Universal Robots PolyScope program: andrea14.urp

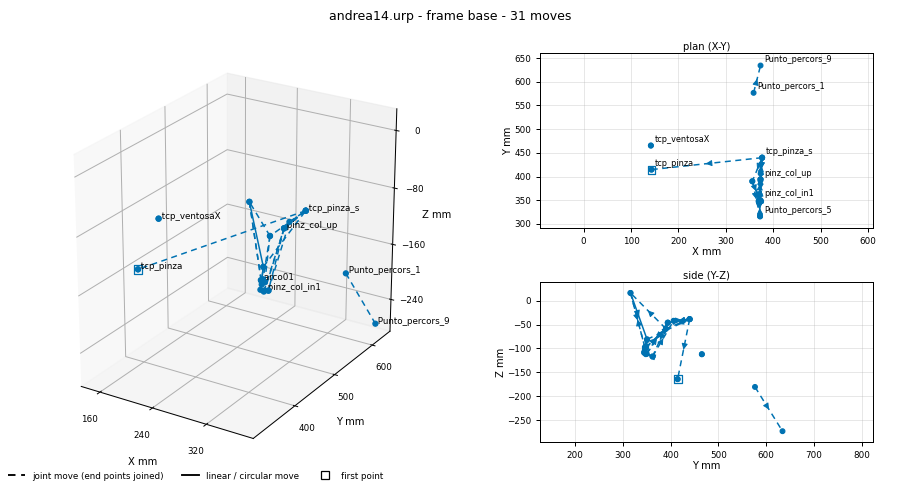
[picture p0: tool path of andrea14.urp in frame base, 31 of 53 moves have a stored position in this frame; points joined in program order, loops and branches not executed]
Program andrea14 (installation=Kong_install12 directory=/programs/usbdisk/andrea14 createdIn=3.15.4.106291 lastSavedIn=3.15.4.106291 robotSerialNumber=2017357596)
Calibrated DH parameters: a=[0.000104, -0.381245, -0.385946, 0.00002, 0.000083, 0]; d=[0.089177, 59.99214, -36.297918, -23.584132, 0.094784, 0.082552]; alpha=[1.570197, -0.003145, 0.002952, 1.570494, -1.570091, 0]; deltaTheta=[-0.00001, -0.459739, 0.638868, -0.17972, -0.000006, -0.000462]
InitVariablesNode variables(variable(name=XY, expression=[0,0]), variable(name=ant, expression=3), variable(name=col, expression=4), variable(name=dump, expression=5), variable(name=ghr, expression=2), variable(name=nCycle, expression=0), variable(name=nfc, expression=1), variable(name=pallStocks, expression=[16,16,16,40,16,16,16,40,16,16,16,40,16,40,0,0,0,0,0,0,0,0,0,0]), variable(name=pick, expression=[0,0]))
Robot Program (runOnlyOnce=false)
  Script file /programs/Kong/relPose.script
    | def relPose(FeaturePose,vect):
    | 
    |     # FeaturePose is the pose for the feature
    |     # vect = p[0.1, 0, 0, 0, 0, 0] makes us move 10cm in the X direction of the feature
    |     # credits: https://forum.universal-robots.com/t/move-tcp-relative-to-feature/15492
    | 
    |    PoseRelativeToFeature = pose_trans(pose_inv(FeaturePose), get_actual_tcp_pose())
    |    MoveTCPRelativeToFeature = pose_add(PoseRelativeToFeature, vect)
    |    return pose_trans(FeaturePose, MoveTCPRelativeToFeature)
    | 
    | end
  Script file /programs/Kong/totf.script_bak
    | def totf(tcpf):
    | 
    |     return sqrt(tcpf[0]*tcpf[0]+tcpf[1]*tcpf[1]+tcpf[2]*tcpf[2]+tcpf[3]*tcpf[3]+tcpf[4]*tcpf[4]+tcpf[5]*tcpf[5])
    | 
    | end
  Script file /programs/Kong/tcpMov.script
    | def tcpMov(vect):
    | 
    |     # FeaturePose is the pose for the feature
    |     # vect = p[0.1, 0, 0, 0, 0, 0] makes us move 10cm in the X direction of the feature
    |     # credits: https://forum.universal-robots.com/t/move-tcp-relative-to-feature/15492
    | 
    |    tcp_pose = get_actual_tcp_pose()
    |    return pose_add(tcp_pose, vect)
    | 
    | 
    | end
  Script file /programs/Kong/calcItemPosition.script_bak
    | def calcItemPosition(pick, item, pallDefs, grid, featOrigin):
    | 
    |     # calcola la posizione assoluta del pezzo scelto da pickPalletItem
    | 
    |     # nPosX è il numero di colonne
    |     # nPosY è il numero di righe
    |     # distX è la distanza tra colonne
    |     # distY è la distanza tra righe
    |     # [posX1, posY1] è la posizione del primo pezzo rispetto all'origine del pallet
    | 
    |     nPallet = pick[0] + 1 # numero del pallet (gli id partono da 0)
    |     nItem = pick[1] + 1 # numero del pezzo
    | 
    |     nPosXgrid = grid[0] # numero di posizioni della giglia in X
    |     distXgrid = grid[2] # distanza tra gli slot della griglia in X
    |     distYgrid = grid[3] # distanza tra gli slot della griglia in Y
    | 
    |     pallPosX = nPallet%nPosXgrid
    |     if(pallPosX==0): pallPosX = nPosXgrid end
    |     pallPosY = ceil(nPallet/nPosXgrid)
    | 
    |     pallPosX1 = grid[4]
    |     pallPosY1 = grid[5]
    | 
    | 
    |     nPosX = pallDefs[item,0]
    |     nPosY = pallDefs[item,1]
    |     distX = pallDefs[item,2]
    |     distY = pallDefs[item,3]
    |     posX1 = pallDefs[item,4]
    |     posY1 = pallDefs[item,5]
    | 
    |     posX = nItem%nPosX
    |     if(posX==0): posX = nPosX end
    |     posY = ceil(nItem/nPosX)
    | 
    |     # [X,Y] è la posizione del pezzo rispetto all'origine della griglia
    | 
    |     X=distX*(posX - 1) + posX1 + distXgrid*(pallPosX - 1) + pallPosX1
    |     Y=distY*(posY - 1) + posY1 + distYgrid*(pallPosY - 1) + pallPosY1
    |     xy=[X,Y]
    | 
    |     return xy
    | 
    |  end
  Script file /programs/usbdisk/andrea8/pickPalletItem.script
    | def pickPalletItem(type, pallDefs, pallTypes, pallStocks):
    | 
    |   # seleziona un pezzo sulla griglia, noti il tipo di pezzo e lo stato della griglia
    | 
    |   # lo script funziona finché le variabili del robot non vengono resettate. Tuttavia, anche
    |   # in caso di riavvio, è possibile scrivere manualmente le info sulla griglia e lo stock
    |   # all'inizio del programma, così da 'insegnare' al robot dove farlo
    |   # riprendere
    | 
    |   iPallet = 0 # inizializzo l'id del pallet
    | 
    |   while iPallet < length(pallStocks):
    | 
    |     if pallTypes[iPallet] == type and pallStocks[iPallet] > 0 :
    | 
    |       nItems = pallStocks[iPallet] # numero di pezzi nello stock del pallet iesimo
    | 
    |       nPosX = pallDefs[type,0] # numero di posizioni lungo x, come definito per il pallet di tipo "type"
    |       nPosY = pallDefs[type,1] # numero di posizioni lungo y, come definito per il pallet di tipo "type"
    | 
    |       stockMax = nPosX*nPosY
    |       iItem = stockMax - nItems # id del pezzo
    | 
    |       pick = [iPallet,iItem]
    | 
    |       # pick = [id del pallet, id del pezzo]
    | 
    |       return pick
    |  end
    | iPallet = iPallet + 1
    | end
    | end
  Script file /home/ur/ursim-current/programs/andrea11/stockUpdate.script_bak
    | def stockUpdate(pick,stock):
    | 
    |     # simple function that ingests the output of pickItem and returns the
    |     # modified stock array. just so to avoid using global variables and
    |     # multi-dimensional arrays
    | 
    |     i = pick[0]
    |     stock[i] = stock[i] - 1
    |     return stock
    | 
    | 
    | end
  Script file /programs/Kong/ini_grid.script_bak.script
    | def ini_grid():
    | 
    |     # grid = [nPallPosX, nPallPosY, distPallX, distPallY, pallPosX1, pallPosY1, pallPosZ1]
    |     # la struttura e' del tutto analoga in logica con quella espressa in defs
    |     grid = [4, 4, 90, 90, 10, 20, 6]
    |     return grid
    | end
  Script file /programs/Kong/ini_defs.script
    | def ini_defs():
    | 
    |     # definition = [nPosX,nPosY,distX,distY,posX1,posY1,posZ1]
    | 
    |     # nPosX è il numero di colonne
    |     # nPosY è il numero di righe
    |     # distX è la distanza tra colonne
    |     # distY è la distanza tra righe
    |     # [posX1, posY1] è la posizione del primo pezzo rispetto all'origine del pallet
    |     # posZ1 e' la posizione che deve raggiungere il TCP lungo asse Z, che sarebbe asse verticale
    | 
    |     defs = [
    |         [0, 0, 0, 0, 0, 0, 0], # slot vuoto
    |         [4, 10, 18, 8, 12, 7.4, 9.1], # pallet nfc
    |         [4, 4, 21, 21, 8.2, 7.5, 50], # pallet ghiere
    |         [1, 1, 0, 0, 132.06, 44, 16.05], # stazione antenna
    |         [1, 2, 0, 40, 20.256, 24, 27.85], # stazione incollaggio
    |         [1, 1, 0, 0, 40, 40, 50] # cestino
    |     ]
    |     return defs
    | end
  Script file /programs/Kong/ini_types.script_bak_bak
    | def ini_types():
    | 
    |     visualTypes = [
    | 
    |         [0, 0, 0, 0],
    |         [0, 0, 0, 0],
    |         [0,0,0,0],
    |         [0,0,0,0],
    |         [0,ghr,0,nfc],
    |         [dump,0,0,0]
    | 
    |     ]
    | 
    | # purtroppo fare questa array vuota di dimensione (righe)x(colonne) per aggirare le limitazioni di UR
    | # bisogna ricordarsi di cambiare questa dichiarazione di types se si cambia dimensione griglia
    | 
    |      types = [0,0,0,0,0,0,0,0,0,0,0,0,0,0,0,0,0,0,0,0,0,0,0,0]
    | 
    |     iii = 0
    |     s = size(visualTypes)
    |     i = 0
    |     while i < s[0]:
    | 
    |         ii=0
    |         while ii < s[1]:
    | 
    |             types[iii] = visualTypes[s[0]-1-i,ii]
    |             ii = ii + 1
    |             iii = iii + 1
    |         end
    |     i = i + 1
    |     end
    |     return types
    | end
  Script file /programs/Kong/ini_stocks2.script
    | def ini_stocks(defs, types):
    | 
    |     global f = -1 # usa questo carattere per inizializzare automaticamente pallet pieni
    | 
    |     visualStocks = [
    | 
    |         [f, f, f, f],
    |         [f, f, f, f],
    |         [f, f, f, f],
    |         [f, f, f, f],
    |         [f, f, f, 27],
    |         [f ,f, f, f]
    | 
    |     ]
    | 
    | # purtroppo fare questa array vuota di dimensione (righe)x(colonne) per aggirare le limitazioni di UR
    | # bisogna ricordarsi di cambiare questa dichiarazione di types se si cambia dimensione griglia
    | 
    |      stocks = [0,0,0,0,0,0,0,0,0,0,0,0,0,0,0,0,0,0,0,0,0,0,0,0]
    | 
    |     iii = 0
    |     s = size(visualStocks)
    |     i = 0
    |     while i < s[0]:
    | 
    |         ii=0
    |         while ii < s[1]:
    |             if visualStocks[s[0]-1-i,ii] == f:
    |                 nPosX = defs[types[iii], 0]
    |                 nPosY = defs[types[iii], 1]
    |                 stocks[iii] = nPosX*nPosY
    |             else:
    | 
    |                 stocks[iii] = visualStocks[s[0]-1-i,ii]
    |             end
    |             ii = ii + 1
    |             iii = iii + 1
    |         end
    |     i = i + 1
    |     end
    |     return stocks
    | end
  Script file /programs/Kong/gen_tcp_grid.script
    | def next_tcp_grid_pos(cur_pos,size,dist):
    | 
    | # size e' la dimensione della griglia da generare,
    | # 2 significa 2x2, 3 significa 3x3 etc
    | 
    | rel_p = [0,0]
    | tcpp = get_actual_tcp_pose()
    | 
    | posX = cur_pos%size
    | if(posX==0): posX = size end
    | posY = ceil(cur_pos/size)
    | 
    | actual_dx = -dist*(size-1)/2 + (posX-1)*dist
    | actual_dy= -dist*(size-1)/2 + (posY-1)*dist
    | 
    | posX = (cur_pos+1)%size
    | if(posX==0): posX = size end
    | posY = ceil((cur_pos+1)/size)
    | 
    | next_dx = -dist*(size-1)/2 + (posX-1)*dist
    | next_dy= -dist*(size-1)/2 + (posY-1)*dist
    | 
    | rel_p = [next_dx - actual_dx, next_dy - actual_dy]
    | 
    | return rel_p
    | 
    | end
  If nCycle≟0
    Set DigitalOutput pin=digital_out[1]; digitalValue=0
    Set DigitalOutput pin=digital_out[0]; digitalValue=0
    pallTypes := ini_types()
    nfc_ck_override := True
    grid := ini_grid()
    pallDefs := ini_defs()
    pallStocks := ini_stocks(pallDefs,pallTypes)
    SuppressedNode
      Popup Message (haltProgram=false inputType=Variable) variable=grid
    ghr := ghr
    nfc := nfc
    ant := ant
    col := col
    dump := dump
    URCap Close Gripper (SCHUNK End-of-Arm Modular System for UR, SCHUNK GmbH & Co.)
    nCycle := 1
    nfc_check := False
    ghr_check := False
    cmp_x_in := 0
    cmp_y_in := 0
    cmp_x_out := 0
    cmp_y_out := 0
    cmp_x := False
    cmp_y := False
    Wait Sleep waitTime=1
  MoveJ speed 60 deg/s, acceleration 80 deg/s^2 (useActiveTCP=false) tcp=Pinza
    Waypoint tcp_pinza: TCP in base x=143.254 y=414.593 z=-164.379 mm, rx=-2.3787 ry=0.7213 rz=1.7106 rad; joints [-127.002, -49.901, 105.969, -114.073, -24.505, -23.784] deg; flange x=184.208 y=554.939 z=9.914 mm, rx=-2.3787 ry=0.7213 rz=1.7106 rad
    item := ghr
    pick := pickPalletItem(item,pallDefs,pallTypes,pallStocks)
    lastpick := pick
    SuppressedNode
      Popup Message (haltProgram=false inputType=Variable) variable=pick
    XY := calcItemPosition(pick, item,pallDefs, grid,piano_moduli)
    p_pall := relPose(piano_moduli,p[(XY[0]+cmp_x_in)/1000,(XY[1]+cmp_y_in)/1000,0.0,0.0,0.0,0.0])
    SuppressedNode
      Popup Message (haltProgram=false inputType=Variable) variable=XY
    Waypoint Punto_percors (Variable): motionParameters(blendRadius=0.004); variable=p_pall
  MoveL speed 250 mm/s, acceleration 1200 mm/s^2 (useActiveTCP=false) tcp=Pinza; feature=Base
    MoveDirectionNode (selectedDirection=ZMinus toolParams=0.05, 1.2) feature=origine_moduli
      Until DISTANCE (allowActions=true deceleration=3 distanceNodeType=STOP) Distance=0.1; motionParameters(blendRadius=0)
        URCap Open Gripper (SCHUNK End-of-Arm Modular System for UR, SCHUNK GmbH & Co.)
        p_pezzo := relPose(piano_moduli,p[0.0, 0.0, 125/1000, 0.0, 0.0, 0.0])
        Waypoint Punto_percors (Variable): variable=p_pezzo
        pallStocks := stockUpdate(pick,pallStocks)
        cmp_x := False
        cmp_y := False
      Until EXPRESSION (allowActions=true) ExpressionBranch=totf(get_tcp_force())>92
        ghr_check := False
        ghr_attpt := 0
        cmp_x := True
        Loop While (checkContinuously=false) expression=ghr_check≟ False
          SuppressedNode
            MoveL speed 125 mm/s, acceleration 600 mm/s^2 (useActiveTCP=false) tcp=Pinza; feature=Base
              p_pezzo := relPose(piano_moduli,p[0.0, 0.0, -125*0.001, 0.0, 0.0, 0.0])
              Waypoint Punto_percors (Variable): variable=p_pezzo
              URCap Open Gripper (SCHUNK End-of-Arm Modular System for UR, SCHUNK GmbH & Co.)
              p_pezzo := relPose(piano_moduli,p[0.0, 0.0, 125/1000, 0.0, 0.0, 0.0])
              Waypoint Punto_percors (Variable): variable=p_pezzo
              pallStocks := stockUpdate(pick,pallStocks)
              SuppressedNode
                Popup Message (haltProgram=false inputType=Variable) variable=pallStocks
          ghr_attpt := ghr_attpt+1
          MoveL speed 125 mm/s, acceleration 600 mm/s^2 (useActiveTCP=false) tcp=Pinza; feature=Base
            Waypoint Punto_percor_14 (Relative): relativeFromPosition TCP in base x=29.478 y=440.875 z=-307.868 mm, rx=-2.3716 ry=0.6969 rz=1.6945 rad; joints [-115.757, -28.156, 105.846, -162.962, -20.903, 4.096] deg; TCP in base x=29.576 y=447.944 z=-300.79 mm, rx=-2.3716 ry=0.6967 rz=1.6945 rad; joints [-115.45, -28.728, 105.08, -162.418, -20.875, 4.938] deg; flange x=68.514 y=584.323 z=-122.922 mm, rx=-2.3716 ry=0.6967 rz=1.6945 rad
          If ghr_attpt≟8
            ghr_attpt := 0
            cmp_y := True
            MoveL speed 50 mm/s, acceleration 500 mm/s^2 (useActiveTCP=false) tcp=Pinza; feature=Base
              Waypoint Punto_percor_15 (Relative): relativeFromPosition TCP in base x=141.409 y=424.504 z=-142.092 mm, rx=-2.3788 ry=0.7214 rz=1.7106 rad; joints [-126.265, -51.639, 104.635, -112.37, -24.118, -22.276] deg; TCP in base x=142.404 y=430.165 z=-147.7 mm, rx=-2.3787 ry=0.7215 rz=1.7107 rad; joints [-126.02, -50.501, 103.739, -113.086, -23.994, -21.754] deg; flange x=183.37 y=570.533 z=26.574 mm, rx=-2.3787 ry=0.7215 rz=1.7107 rad
          MoveL speed 50 mm/s, acceleration 500 mm/s^2 (useActiveTCP=false) tcp=Pinza; feature=Base
            Waypoint Punto_percor_10 (Relative): relativeFromPosition TCP in base x=141.556 y=430.223 z=-147.722 mm, rx=-2.3788 ry=0.7212 rz=1.7106 rad; joints [-125.948, -50.518, 103.824, -113.299, -23.962, -21.607] deg; TCP in base x=141.537 y=429.491 z=-147.044 mm, rx=-2.3788 ry=0.7213 rz=1.7106 rad; joints [-125.989, -50.655, 103.927, -113.183, -23.981, -21.693] deg; flange x=182.477 y=569.847 z=27.245 mm, rx=-2.3788 ry=0.7213 rz=1.7106 rad
          MoveDirectionNode (selectedDirection=ZMinus toolParams=0.05, 1.2) feature=origine_moduli
            Until DISTANCE (allowActions=true deceleration=3 distanceNodeType=STOP) Distance=0.017; motionParameters(blendRadius=0)
              URCap Open Gripper (SCHUNK End-of-Arm Modular System for UR, SCHUNK GmbH & Co.)
              p_pezzo := relPose(piano_moduli,p[0.0, 0.0, 125/1000, 0.0, 0.0, 0.0])
              Waypoint Punto_percors (Variable): variable=p_pezzo
              pallStocks := stockUpdate(pick,pallStocks)
              ghr_check := True
            Until EXPRESSION (allowActions=true) ExpressionBranch=totf(get_tcp_force())>80
              MoveL speed 50 mm/s, acceleration 500 mm/s^2 (useActiveTCP=true) feature=Base
                Waypoint Punto_percors_6 (Relative): relativeFromPosition TCP in base x=4.07 y=674.667 z=69.754 mm, rx=1.9149 ry=-1.1485 rz=-1.8457 rad; joints [-112.275, -36.345, 91.167, -133.706, -10.047, 30.658] deg; TCP in base x=4.143 y=678.166 z=73.281 mm, rx=1.9147 ry=-1.1486 rz=-1.8457 rad; joints [-112.167, -36.367, 90.585, -133.706, -10.021, 31.279] deg; flange x=70.38 y=685.456 z=-8.016 mm, rx=1.9147 ry=-1.1486 rz=-1.8457 rad
  SuppressedNode
    If cmp_x≟ True removedSiblings(If(type=Else checkContinuously=false, children(Assignment(valueSource=Expression, variable=cmp_x_in, expression=cmp_x_in+1))))
      cmp_x_in := cmp_x_in-1
  SuppressedNode
    If cmp_y≟ True removedSiblings(If(type=Else checkContinuously=false, children(Assignment(valueSource=Expression, variable=cmp_y_in, expression=cmp_y_in+1))))
      cmp_y_in := cmp_y_in-1
  nfc_check := False
  Loop While (checkContinuously=false) expression=nfc_check≟ False
    MoveJ speed 60 deg/s, acceleration 80 deg/s^2 (useActiveTCP=false) tcp=Ventosa
      Waypoint tcp_ventosaX: TCP in base x=141.964 y=465.304 z=-112.234 mm, rx=-2.2905 ry=-0.5963 rz=-0.2623 rad; joints [-121.653, -49.489, 100.632, -2.161, 68.856, 127.498] deg; flange x=142.46 y=500.184 z=-13.074 mm, rx=-2.2905 ry=-0.5963 rz=-0.2623 rad
      item := dump
      pick := pickPalletItem(item,pallDefs,pallTypes,pallStocks)
      SuppressedNode
        Popup Message (haltProgram=false inputType=Variable) variable=pick
      XY := calcItemPosition(pick, item,pallDefs, grid,piano_moduli)
      p_pall := relPose(piano_moduli,p[XY[0]/1000,XY[1]/1000,0.0,0.0,0.0,0.0])
      SuppressedNode
        Popup Message (haltProgram=false inputType=Variable) variable=XY
      Waypoint Punto_percors (Variable): motionParameters(blendRadius=0.005); variable=p_pall
      Set DigitalOutput pin=digital_out[0]; digitalValue=0
    MoveJ speed 60 deg/s, acceleration 80 deg/s^2 (useActiveTCP=false) tcp=Ventosa
      Waypoint tcp_ventosaX: TCP in base x=141.964 y=465.304 z=-112.234 mm, rx=-2.2905 ry=-0.5963 rz=-0.2623 rad; joints [-121.653, -49.489, 100.632, -2.161, 68.856, 127.498] deg; flange x=142.46 y=500.184 z=-13.074 mm, rx=-2.2905 ry=-0.5963 rz=-0.2623 rad
      SuppressedNode
        Waypoint tcp_ventosaY_s: TCP in base x=355.984 y=389.916 z=-58.857 mm, rx=-1.401 ry=-1.0647 rz=1.3858 rad; joints [-146.472, -36.177, 73.345, -37.097, -55.375, 194.745] deg; pose in feature x=141.985 y=465.345 z=-112.215 mm, rx=-1.4011 ry=-1.0646 rz=1.3857 rad; flange x=401.93 y=456.119 z=8.64 mm, rx=-1.401 ry=-1.0647 rz=1.3858 rad
      item := nfc
      pick := pickPalletItem(item,pallDefs,pallTypes,pallStocks)
      SuppressedNode
        Popup Message (haltProgram=false inputType=Variable) variable=pick
      XY := calcItemPosition(pick, item,pallDefs, grid,piano_moduli)
      p_pall := relPose(piano_moduli,p[XY[0]/1000,XY[1]/1000,0.0,0.0,0.0,0.0])
      SuppressedNode
        Popup Message (haltProgram=false inputType=Variable) variable=XY
      Waypoint Punto_percors (Variable): variable=p_pall
      p_pezzo := relPose(piano_moduli,p[0.0, 0.0, -170*0.001, 0.0, 0.0, 0.0])
      Waypoint Punto_percors (Variable): variable=p_pezzo
      Set DigitalOutput pin=digital_out[0]; digitalValue=1
    Loop Counting (count=3) loopVariable(name=Ciclo_4)
      MoveL speed 1.5 mm/s, acceleration 5 mm/s^2 (useActiveTCP=false) tcp=Ventosa; feature=Base
        p_pezzo := relPose(piano_moduli,p[0.0, 0.0, -12*0.001, 0.0, 0.0, 0.0])
        Waypoint Punto_percors (Variable): variable=p_pezzo
        Wait Sleep waitTime=4
        p_pezzo := relPose(piano_moduli,p[0.0, 0.0, 12/1000, 0.0, 0.0, 0.0])
        Waypoint Punto_percors (Variable): variable=p_pezzo
        SuppressedNode
          Popup Message (haltProgram=false inputType=Variable) variable=pallStocks
    pallStocks := stockUpdate(pick,pallStocks)
    MoveJ speed 60 deg/s, acceleration 80 deg/s^2 (useActiveTCP=true)
      Waypoint Punto_percor_17 (Relative): relativeFromPosition TCP in base x=284.521 y=550.156 z=-280.841 mm, rx=-2.2786 ry=-0.6987 rz=-0.1736 rad; joints [-129.352, -17.294, 64.16, 9.308, 60.336, 116.033] deg; TCP in base x=285.519 y=620.503 z=-209.796 mm, rx=-2.2786 ry=-0.6987 rz=-0.1734 rad; joints [-125.512, -17.144, 49.814, 21.783, 62.478, 119.625] deg; flange x=285.39 y=658.018 z=-111.601 mm, rx=-2.2786 ry=-0.6987 rz=-0.1734 rad
    MoveJ speed 60 deg/s, acceleration 80 deg/s^2 (useActiveTCP=false) tcp=Ventosa
      Waypoint Punto_percors_1: motionParameters(blendRadius=0.005); TCP in base x=358.691 y=576.543 z=-180.701 mm, rx=-2.2887 ry=-0.6045 rz=-0.2628 rad; joints [-132.678, -21.575, 54.335, 20.288, 61.783, 117.598] deg; flange x=358.684 y=611.454 z=-81.55 mm, rx=-2.2887 ry=-0.6045 rz=-0.2628 rad
      Waypoint Punto_percors_9: TCP in base x=373.356 y=634.147 z=-273.366 mm, rx=-2.2782 ry=-0.6995 rz=-0.1742 rad; joints [-130.565, 2.612, 17.324, 36.849, 59.589, 114.737] deg; flange x=373.138 y=671.629 z=-175.158 mm, rx=-2.2782 ry=-0.6995 rz=-0.1742 rad
    MoveL speed 125 mm/s, acceleration 600 mm/s^2 (useActiveTCP=false) tcp=Ventosa; feature=Base
      p_pezzo := relPose(piano_moduli,p[0.0, 0.0, -60*0.001, 0.0, 0.0, 0.0])
      Waypoint Punto_percors (Variable): variable=p_pezzo
      SuppressedNode
        Wait Sleep waitTime=2.5
      If nfc_ck_override≟ True
        nfc_check := True
      Loop Counting (count=5) loopVariable(name=Ciclo_2)
        Wait Sleep waitTime=0.5
        If digital_in[4]≟ True
          nfc_check := True
      p_pezzo := relPose(piano_moduli,p[0.0, 0.0, 40/1000, 0.0, 0.0, 0.0])
      Waypoint Punto_percors (Variable): variable=p_pezzo
  MoveJ speed 60 deg/s, acceleration 80 deg/s^2 (useActiveTCP=false) tcp=Pinza
    Waypoint tcp_pinza_s: TCP in base x=376.73 y=439.705 z=-38.836 mm, rx=1.938 ry=-1.1644 rz=-1.0826 rad; joints [-133.252, -18.324, 41.242, -57.827, -54.828, 0.25] deg; flange x=407.104 y=665.044 z=-46.064 mm, rx=1.938 ry=-1.1644 rz=-1.0826 rad
    Waypoint pinz_col_up: TCP in base x=373.333 y=393.978 z=-46.215 mm, rx=1.9378 ry=-1.1643 rz=-1.0825 rad; joints [-135.374, -23.969, 54.366, -64.485, -56.557, -1.187] deg; flange x=403.682 y=619.319 z=-53.485 mm, rx=1.9378 ry=-1.1643 rz=-1.0825 rad
    Waypoint pinz_col_in1: TCP in base x=373.185 y=350.07 z=-111.439 mm, rx=1.859 ry=-1.2139 rz=-0.9382 rad; joints [-137.407, -19.377, 60.953, -74.216, -62.773, 4.123] deg; flange x=401.803 y=572.572 z=-149.211 mm, rx=1.859 ry=-1.2139 rz=-0.9382 rad
    URCap Close Gripper (SCHUNK End-of-Arm Modular System for UR, SCHUNK GmbH & Co.)
    Waypoint pinz_col_out: TCP in base x=371.134 y=362.077 z=-117.035 mm, rx=1.8499 ry=-1.2119 rz=-0.9092 rad; joints [-136.429, -17.422, 58.359, -73.529, -63.149, 5.469] deg; flange x=397.507 y=583.951 z=-159.802 mm, rx=1.8499 ry=-1.2119 rz=-0.9092 rad
    SuppressedNode
      Waypoint pinz_col_up: TCP in base x=353.537 y=408.471 z=-60.29 mm, rx=1.9378 ry=-1.1643 rz=-1.0825 rad; joints [-133.591, -22.853, 54.464, -66.388, -55.09, 0.038] deg; flange x=383.886 y=633.812 z=-67.559 mm, rx=1.9378 ry=-1.1643 rz=-1.0825 rad
    Waypoint Punto_percors_2: TCP in base x=373.559 y=406.189 z=-42.147 mm, rx=1.8482 ry=-1.2116 rz=-0.904 rad; joints [-134.183, -19.68, 50.23, -63.704, -61.475, 6.948] deg; flange x=399.547 y=627.929 z=-85.834 mm, rx=1.8482 ry=-1.2116 rz=-0.904 rad
    SuppressedNode
      URCap Open Gripper (SCHUNK End-of-Arm Modular System for UR, SCHUNK GmbH & Co.)
    Waypoint tcp_pinza_s: TCP in base x=376.73 y=439.705 z=-38.836 mm, rx=1.938 ry=-1.1644 rz=-1.0826 rad; joints [-133.252, -18.324, 41.242, -57.827, -54.828, 0.25] deg; flange x=407.104 y=665.044 z=-46.064 mm, rx=1.938 ry=-1.1644 rz=-1.0826 rad
  MoveJ speed 60 deg/s, acceleration 80 deg/s^2 (useActiveTCP=false) tcp=Dosatore_Colla
    Waypoint tcp_coll_s: TCP in base x=355.98 y=389.944 z=-58.821 mm, rx=-0.0221 ry=-3.1138 rz=0.4025 rad; joints [-139.164, -64.295, 106.354, -122.012, -100.828, 102.957] deg; flange x=356.623 y=435.2 z=113.328 mm, rx=0.7684 ry=-2.9515 rz=0.3801 rad
    Waypoint Punto_percors_7: TCP in base x=371.412 y=348.681 z=-96.843 mm, rx=-0.0219 ry=-3.114 rz=0.4022 rad; joints [-143.466, -62.52, 111.583, -129.872, -101.561, 98.637] deg; flange x=372.023 y=393.908 z=75.314 mm, rx=0.7687 ry=-2.9516 rz=0.3799 rad
    Waypoint Punto_percors_8: TCP in base x=371.364 y=346.005 z=-102.454 mm, rx=-0.022 ry=-3.1138 rz=0.4026 rad; joints [-143.686, -62.081, 112.082, -130.84, -101.607, 98.424] deg; flange x=371.995 y=391.277 z=69.691 mm, rx=0.7686 ry=-2.9515 rz=0.3802 rad
    Waypoint Punto_percors_7: TCP in base x=371.412 y=348.681 z=-96.843 mm, rx=-0.0219 ry=-3.114 rz=0.4022 rad; joints [-143.466, -62.52, 111.583, -129.872, -101.561, 98.637] deg; flange x=372.023 y=393.908 z=75.314 mm, rx=0.7687 ry=-2.9516 rz=0.3799 rad
    SuppressedNode
      Waypoint tcp_colla: TCP in base x=141.953 y=465.356 z=-112.213 mm, rx=-0.0207 ry=-2.9002 rz=1.1933 rad; joints [-112.251, -46.475, 88.048, -88.757, -104.681, 134.691] deg; flange x=143.75 y=590.738 z=14.373 mm, rx=0.6882 ry=-2.6438 rz=1.0836 rad
  MoveL speed 250 mm/s, acceleration 1200 mm/s^2 (useActiveTCP=false) tcp=Dosatore_Colla; feature=Base
    Waypoint arco01: TCP in base x=369.128 y=347.673 z=-97.886 mm, rx=-0.3054 ry=2.8059 rz=-0.3653 rad; joints [-138.423, -63.732, 122.875, -154.572, -111.742, 88.494] deg; flange x=313.211 y=386.181 z=66.657 mm, rx=-1.0435 ry=2.6885 rz=-0.4726 rad
    Set DigitalOutput pin=digital_out[1]; digitalValue=1
    Wait Sleep waitTime=0.5
    Waypoint Punto_percors_3: TCP in base x=374.619 y=347.76 z=-99.486 mm, rx=-0.4267 ry=-2.7025 rz=0.3458 rad; joints [-150.963, -55.958, 98.583, -106.41, -87.536, 106.756] deg; flange x=446.604 y=379.598 z=60.165 mm, rx=0.2834 ry=-2.6841 rz=0.1927 rad
    Set DigitalOutput pin=digital_out[1]; digitalValue=0
  MoveJ speed 60 deg/s, acceleration 80 deg/s^2 (useActiveTCP=false) tcp=Dosatore_Colla
    Waypoint tcp_coll_s: motionParameters(blendRadius=0.005); TCP in base x=355.98 y=389.944 z=-58.821 mm, rx=-0.0221 ry=-3.1138 rz=0.4025 rad; joints [-139.164, -64.295, 106.354, -122.012, -100.828, 102.957] deg; flange x=356.623 y=435.2 z=113.328 mm, rx=0.7684 ry=-2.9515 rz=0.3801 rad
  MoveJ speed 60 deg/s, acceleration 80 deg/s^2 (useActiveTCP=false) tcp=Ventosa
    SuppressedNode
      Waypoint tcp_ventosaY_s: TCP in base x=355.984 y=389.916 z=-58.857 mm, rx=-1.401 ry=-1.0647 rz=1.3858 rad; joints [-146.472, -36.177, 73.345, -37.097, -55.375, 194.745] deg; flange x=401.93 y=456.119 z=8.64 mm, rx=-1.401 ry=-1.0647 rz=1.3858 rad
    Waypoint Punto_percors_5: TCP in base x=372.347 y=315.923 z=16.067 mm, rx=-1.0185 ry=-1.3146 rz=1.0001 rad; joints [-156.567, -51.004, 84.609, -33.5, -65.468, 164.694] deg; flange x=417.701 y=339.435 z=107.936 mm, rx=-1.0185 ry=-1.3146 rz=1.0001 rad
    Waypoint Punto_percor_11: TCP in base x=370.683 y=345.937 z=-97.463 mm, rx=-1.0185 ry=-1.3145 rz=1.0003 rad; joints [-153.919, -39.647, 83.462, -43.728, -62.813, 164.763] deg; flange x=416.048 y=369.471 z=-5.606 mm, rx=-1.0185 ry=-1.3145 rz=1.0003 rad
    Wait Sleep waitTime=1
    Set DigitalOutput pin=digital_out[0]; digitalValue=0
    Wait Sleep waitTime=1
    Waypoint Punto_percors_5: TCP in base x=372.347 y=315.923 z=16.067 mm, rx=-1.0185 ry=-1.3146 rz=1.0001 rad; joints [-156.567, -51.004, 84.609, -33.5, -65.468, 164.694] deg; flange x=417.701 y=339.435 z=107.936 mm, rx=-1.0185 ry=-1.3146 rz=1.0001 rad
    SuppressedNode
      Waypoint Punto_percors_4: 
  MoveL speed 250 mm/s, acceleration 1200 mm/s^2 (useActiveTCP=false) tcp=Pressa; feature=Base
    Waypoint Punto_percor_12: motionParameters(blendRadius=0.005); TCP in base x=370.755 y=350.619 z=-81.186 mm, rx=0.1982 ry=-1.5625 rz=-0.2205 rad; joints [-152.069, -45.343, 79.221, -33.787, -60.961, 74.712] deg; flange x=416.359 y=391.91 z=78.389 mm, rx=0.1982 ry=-1.5625 rz=-0.2205 rad
    Waypoint Punto_percor_13: TCP in base x=370.688 y=344.213 z=-108.905 mm, rx=0.1982 ry=-1.5625 rz=-0.2205 rad; joints [-152.591, -43.593, 80.784, -37.111, -61.48, 74.725] deg; flange x=416.28 y=385.497 z=50.675 mm, rx=0.1982 ry=-1.5625 rz=-0.2205 rad
    Wait Sleep waitTime=2
    Waypoint Punto_percor_12: TCP in base x=370.755 y=350.619 z=-81.186 mm, rx=0.1982 ry=-1.5625 rz=-0.2205 rad; joints [-152.069, -45.343, 79.221, -33.787, -60.961, 74.712] deg; flange x=416.359 y=391.91 z=78.389 mm, rx=0.1982 ry=-1.5625 rz=-0.2205 rad
    SuppressedNode
      Waypoint tcp_pressaY: TCP in base x=141.469 y=430.16 z=-147.709 mm, rx=-0.2128 ry=-1.5595 rz=0.1907 rad; joints [-127.014, -38.383, 85.876, -47.443, -35.896, 104.766] deg; flange x=188.109 y=545.63 z=-30.49 mm, rx=-0.2128 ry=-1.5595 rz=0.1907 rad
    SuppressedNode
      Waypoint tcp_pressaX: TCP in base x=141.415 y=430.194 z=-147.729 mm, rx=-1.3127 ry=-2.237 rz=-0.9404 rad; joints [-120.759, -49.8, 97.992, 0.536, 69.418, 38.219] deg; flange x=142.623 y=514.321 z=1.167 mm, rx=-1.3127 ry=-2.237 rz=-0.9404 rad
  MoveJ speed 60 deg/s, acceleration 80 deg/s^2 (useActiveTCP=false) tcp=Pinza
    Waypoint tcp_pinza_s: TCP in base x=376.73 y=439.705 z=-38.836 mm, rx=1.938 ry=-1.1644 rz=-1.0826 rad; joints [-133.252, -18.324, 41.242, -57.827, -54.828, 0.25] deg; flange x=407.104 y=665.044 z=-46.064 mm, rx=1.938 ry=-1.1644 rz=-1.0826 rad
    Waypoint pinz_col_up: TCP in base x=373.333 y=393.978 z=-46.215 mm, rx=1.9378 ry=-1.1643 rz=-1.0825 rad; joints [-135.374, -23.969, 54.366, -64.485, -56.557, -1.187] deg; flange x=403.682 y=619.319 z=-53.485 mm, rx=1.9378 ry=-1.1643 rz=-1.0825 rad
    Waypoint pinz_col_out: TCP in base x=371.134 y=362.077 z=-117.035 mm, rx=1.8499 ry=-1.2119 rz=-0.9092 rad; joints [-136.429, -17.422, 58.359, -73.529, -63.149, 5.469] deg; flange x=397.507 y=583.951 z=-159.802 mm, rx=1.8499 ry=-1.2119 rz=-0.9092 rad
    Waypoint pinz_col_in: TCP in base x=373.168 y=347.955 z=-112.194 mm, rx=1.8591 ry=-1.2139 rz=-0.9382 rad; joints [-137.526, -19.49, 61.363, -74.482, -62.872, 4.052] deg; flange x=401.789 y=570.456 z=-149.961 mm, rx=1.8591 ry=-1.2139 rz=-0.9382 rad
    URCap Open Gripper (SCHUNK End-of-Arm Modular System for UR, SCHUNK GmbH & Co.)
    Waypoint pinz_col_up: TCP in base x=373.333 y=393.978 z=-46.215 mm, rx=1.9378 ry=-1.1643 rz=-1.0825 rad; joints [-135.374, -23.969, 54.366, -64.485, -56.557, -1.187] deg; flange x=403.682 y=619.319 z=-53.485 mm, rx=1.9378 ry=-1.1643 rz=-1.0825 rad
    SuppressedNode
      Waypoint pinz_col_up: TCP in base x=353.537 y=408.471 z=-60.29 mm, rx=1.9378 ry=-1.1643 rz=-1.0825 rad; joints [-133.591, -22.853, 54.464, -66.388, -55.09, 0.038] deg; flange x=383.886 y=633.812 z=-67.559 mm, rx=1.9378 ry=-1.1643 rz=-1.0825 rad
    SuppressedNode
      Waypoint Punto_percors_2: TCP in base x=354.064 y=441.822 z=-77.166 mm, rx=1.8482 ry=-1.2116 rz=-0.904 rad; joints [-131.419, -13.619, 42.947, -63.355, -59.194, 8.709] deg; flange x=380.052 y=663.563 z=-120.852 mm, rx=1.8482 ry=-1.2116 rz=-0.904 rad
    SuppressedNode
      URCap Open Gripper (SCHUNK End-of-Arm Modular System for UR, SCHUNK GmbH & Co.)
    Waypoint tcp_pinza_s: TCP in base x=376.73 y=439.705 z=-38.836 mm, rx=1.938 ry=-1.1644 rz=-1.0826 rad; joints [-133.252, -18.324, 41.242, -57.827, -54.828, 0.25] deg; flange x=407.104 y=665.044 z=-46.064 mm, rx=1.938 ry=-1.1644 rz=-1.0826 rad
  MoveJ speed 60 deg/s, acceleration 80 deg/s^2 (useActiveTCP=false) tcp=Pinza
    Waypoint tcp_pinza: TCP in base x=143.254 y=414.593 z=-164.379 mm, rx=-2.3787 ry=0.7213 rz=1.7106 rad; joints [-127.002, -49.901, 105.969, -114.073, -24.505, -23.784] deg; flange x=184.208 y=554.939 z=9.914 mm, rx=-2.3787 ry=0.7213 rz=1.7106 rad
    SuppressedNode
      Popup Message (haltProgram=false inputType=Variable) variable=pick
    item := ghr
    XY := calcItemPosition(lastpick, item,pallDefs, grid,piano_moduli)
    p_pall := relPose(piano_moduli,p[XY[0]/1000-0.001,XY[1]/1000,0.0,0.0,0.0,0.0])
    SuppressedNode
      Popup Message (haltProgram=false inputType=Variable) variable=XY
    Waypoint Punto_percors (Variable): variable=p_pall
  MoveL speed 250 mm/s, acceleration 1200 mm/s^2 (useActiveTCP=false) tcp=Pinza; feature=Base
    MoveDirectionNode (selectedDirection=ZMinus toolParams=0.05, 1.2) feature=origine_moduli
      Until DISTANCE (allowActions=true deceleration=3 distanceNodeType=STOP) Distance=0.085; motionParameters(blendRadius=0)
        URCap Close Gripper (SCHUNK End-of-Arm Modular System for UR, SCHUNK GmbH & Co.)
        p_pezzo := relPose(piano_moduli,p[0.0, 0.0, 125/1000, 0.0, 0.0, 0.0])
        Waypoint Punto_percors (Variable): variable=p_pezzo
        SuppressedNode
          pallStocks := stockUpdate(pick,pallStocks)
        cmp_x := False
        cmp_y := False
      Until EXPRESSION (allowActions=true) ExpressionBranch=totf(get_tcp_force())>95
        ghr_check := False
        ghr_attpt := 0
        cmp_x := True
        Loop While (checkContinuously=false) expression=ghr_check≟ False
          SuppressedNode
            MoveL speed 125 mm/s, acceleration 600 mm/s^2 (useActiveTCP=false) tcp=Pinza; feature=Base
              p_pezzo := relPose(piano_moduli,p[0.0, 0.0, -125*0.001, 0.0, 0.0, 0.0])
              Waypoint Punto_percors (Variable): variable=p_pezzo
              URCap Open Gripper (SCHUNK End-of-Arm Modular System for UR, SCHUNK GmbH & Co.)
              p_pezzo := relPose(piano_moduli,p[0.0, 0.0, 125/1000, 0.0, 0.0, 0.0])
              Waypoint Punto_percors (Variable): variable=p_pezzo
              pallStocks := stockUpdate(pick,pallStocks)
              SuppressedNode
                Popup Message (haltProgram=false inputType=Variable) variable=pallStocks
          ghr_attpt := ghr_attpt+1
          MoveL speed 125 mm/s, acceleration 600 mm/s^2 (useActiveTCP=false) tcp=Pinza; feature=Base
            Waypoint Punto_percor_16 (Relative): relativeFromPosition TCP in base x=21.48 y=497.646 z=-275.999 mm, rx=-2.3783 ry=0.7214 rz=1.7109 rad; joints [-112.781, -28.123, 96.79, -160.334, -20.71, 12.471] deg; TCP in base x=21.716 y=511.71 z=-261.76 mm, rx=-2.3784 ry=0.7216 rz=1.7108 rad; joints [-112.302, -28.904, 94.899, -158.934, -20.726, 13.834] deg; flange x=62.735 y=652.049 z=-87.475 mm, rx=-2.3784 ry=0.7216 rz=1.7108 rad
          If ghr_attpt≟4
            ghr_attpt := 1
            cmp_y := True
            MoveL speed 50 mm/s, acceleration 500 mm/s^2 (useActiveTCP=false) tcp=Pinza; feature=Base
              Waypoint Punto_percor_15 (Relative): relativeFromPosition TCP in base x=141.409 y=424.504 z=-142.092 mm, rx=-2.3788 ry=0.7214 rz=1.7106 rad; joints [-126.265, -51.639, 104.635, -112.37, -24.118, -22.276] deg; TCP in base x=142.404 y=430.165 z=-147.7 mm, rx=-2.3787 ry=0.7215 rz=1.7107 rad; joints [-126.02, -50.501, 103.739, -113.086, -23.994, -21.754] deg; flange x=183.37 y=570.533 z=26.574 mm, rx=-2.3787 ry=0.7215 rz=1.7107 rad
          MoveL speed 50 mm/s, acceleration 500 mm/s^2 (useActiveTCP=false) tcp=Pinza; feature=Base
            Waypoint Punto_percor_10 (Relative): relativeFromPosition TCP in base x=141.556 y=430.223 z=-147.722 mm, rx=-2.3788 ry=0.7212 rz=1.7106 rad; joints [-125.948, -50.518, 103.824, -113.299, -23.962, -21.607] deg; TCP in base x=141.537 y=429.491 z=-147.044 mm, rx=-2.3788 ry=0.7213 rz=1.7106 rad; joints [-125.989, -50.655, 103.927, -113.183, -23.981, -21.693] deg; flange x=182.477 y=569.847 z=27.245 mm, rx=-2.3788 ry=0.7213 rz=1.7106 rad
          MoveDirectionNode (selectedDirection=ZMinus toolParams=0.05, 1.2) feature=origine_moduli
            Until DISTANCE (allowActions=true deceleration=3 distanceNodeType=STOP) Distance=0.025; motionParameters(blendRadius=0)
              URCap Close Gripper (SCHUNK End-of-Arm Modular System for UR, SCHUNK GmbH & Co.)
              p_pezzo := relPose(piano_moduli,p[0.0, 0.0, 125/1000, 0.0, 0.0, 0.0])
              Waypoint Punto_percors (Variable): variable=p_pezzo
              SuppressedNode
                pallStocks := stockUpdate(pick,pallStocks)
              ghr_check := True
            Until EXPRESSION (allowActions=true) ExpressionBranch=totf(get_tcp_force())>85
              MoveL speed 50 mm/s, acceleration 500 mm/s^2 (useActiveTCP=true) feature=Base
                Waypoint Punto_percors_6 (Relative): relativeFromPosition TCP in base x=4.07 y=674.667 z=69.754 mm, rx=1.9149 ry=-1.1485 rz=-1.8457 rad; joints [-112.275, -36.345, 91.167, -133.706, -10.047, 30.658] deg; TCP in base x=4.143 y=678.166 z=73.281 mm, rx=1.9147 ry=-1.1486 rz=-1.8457 rad; joints [-112.167, -36.367, 90.585, -133.706, -10.021, 31.279] deg; flange x=70.38 y=685.456 z=-8.016 mm, rx=1.9147 ry=-1.1486 rz=-1.8457 rad
  SuppressedNode
    If cmp_x≟ True removedSiblings(If(type=Else checkContinuously=false, children(Assignment(valueSource=Expression, variable=cmp_x_out, expression=cmp_x_out+1))))
      cmp_x_out := cmp_x_out-1
  SuppressedNode
    If cmp_y≟ True removedSiblings(If(type=Else checkContinuously=false, children(Assignment(valueSource=Expression, variable=cmp_y_out, expression=cmp_y_out+1))))
      cmp_y_out := cmp_y_out-1
  SuppressedNode
    Popup Message (haltProgram=false inputType=Variable) variable=pick
